// ==========================================
// 6. BLOCO MQTT PUBLISH
//    Steps 10/20 -> sPayload (Tool + Status)
//    Steps 30/40 -> sPayloadTools (tempos por máquina)
// ==========================================
IF iStep = 30 OR iStep = 40 THEN
    fbMqttPublish(
        xExecute       := bExecutePublish,
        mqttClient     := fbMqttClient,
        wsTopicName    := wsTopic,
        pbPayload      := ADR(sPayloadTools),
        udiPayloadSize := INT_TO_UDINT(LEN(sPayloadTools)),
        eQoS           := 0,
        xRetain        := FALSE
    );
ELSE
    fbMqttPublish(
        xExecute       := bExecutePublish,
        mqttClient     := fbMqttClient,
        wsTopicName    := wsTopic,
        pbPayload      := ADR(sPayload),
        udiPayloadSize := INT_TO_UDINT(LEN(sPayload)),
        eQoS           := 0,
        xRetain        := FALSE
    );
END_IF

END_PROGRAM
